// TIA Portal project "DPS" (V18)

(* hardware
DEVICE "S7-1200-Station_1"  S7-1200 Station
   slot 0: "Baugruppenträger_0"  S7-1200 Rack  Rack  V1.0
   slot 1: "DPS"  CPU 1215C DC/DC/DC  6ES7 215-1AG40-0XB0  V4.5
*)

// ===== PLC "DPS"  CPU 1215C DC/DC/DC =====

VAR_GLOBAL   // PLC tag table "Lichter"
   "grünLED" AT %Q0.4 : Bool;
   "gelbLED" AT %Q0.5 : Bool;
   "rotLED" AT %Q0.6 : Bool;
   "rotLED_online" AT %Q0.7 : Bool;
END_VAR

VAR_GLOBAL   // PLC tag table "Farbsensor"
   "FarbWert" AT %IW64 : Int;
END_VAR

VAR_GLOBAL   // PLC tag table "WareneingangAusgang"
   "ausgangLS" AT %I0.2 : Bool;
   "eingangLS" AT %I0.3 : Bool;
END_VAR

VAR_GLOBAL   // PLC tag table "KameraHR"
   "refKameraHochRunter" AT %I0.0 : Bool;   // Referenzschalter für den Encoder
   "encoderHR_A" AT %I0.4 : Bool;   // Encoder A
   "encoderHR_B" AT %I0.5 : Bool;   // Encoder B
   "kameraHoch" AT %Q0.0 : Bool;   // Motor drehen um Kamera nach oben zu bewegen
   "kameraRunter" AT %Q0.1 : Bool;   // Motor drehen um Kamera nach unten zu bewegen
   "PWM_kameraHR" AT %QW1000 : Int;   // Prozentualer Wert für die geschwindigkeit des Motors
   "EncoderWertHR" AT %ID1000 : DInt;   // Der Zählwert welche die Position bestimmt
END_VAR

VAR_GLOBAL   // PLC tag table "KameraLR"
   "refKameraLinksRechts" AT %I0.1 : Bool;   // Referenzschalter für den Encoder
   "encoderLR_A" AT %I0.6 : Bool;   // Encoder A
   "encoderLR_B" AT %I0.7 : Bool;   // Encoder B
   "kameraLinks" AT %Q0.2 : Bool;   // Motor drehen um Kamera nach links zu bewegen
   "kameraRechts" AT %Q0.3 : Bool;   // Motor drehen um Kamera nach rechts zu bewegen
   "PWM_kameraLR" AT %QW1002 : Int;   // Prozentualer Wert für die geschwindigkeit des Motors
   "EncoderWertLR" AT %ID1004 : DInt;   // Der Zählwert welche die Position bestimmt
END_VAR

DATA_BLOCK "DB_Global"   // DB1
{ S7_Optimized_Access := 'TRUE' }
VERSION : 0.1
   VAR
      farbwert : Int;
      farbbereich_rot : Bool;
      farbbereich_weiss : Bool;
      farbbereich_blau : Bool;
      input : Bool;
      output : Bool;
      referenziert_X : Bool;
      referenziert_Y : Bool;
      referenzieren : Bool;
      reset : Bool;
      Farbe : Struct
         berechne : Bool;
         rotOben : Int;
         rotUnten : Int;
         weissOben : Int;
         weissUnten : Int;
         blauOben : Int;
         blauUnten : Int;
      END_STRUCT;
   END_VAR
BEGIN
END_DATA_BLOCK

DATA_BLOCK "DB_Referenzen"   // DB2
{ S7_Optimized_Access := 'TRUE' }
VERSION : 0.1
   VAR RETAIN
      Calib : Struct
         Limits : Struct
            grenze_x_oben : DInt := 1700;
            grenze_x_unten : DInt := 0;
            grenze_y_oben : DInt := 700;
            grenze_y_unten : DInt := 0;
         END_STRUCT;
         Positionen : Struct
            Home : Struct
               position_home_X : DInt := 900;
               position_home_Y : DInt := 350;
            END_STRUCT;
            HBW : Struct
               position_hbw_X : DInt := 1500;
               position_hbw_Y : DInt := 250;
            END_STRUCT;
            Parken : Struct
               position_parken_X : DInt := 1000;
               position_parken_Y : DInt := 5;
            END_STRUCT;
         END_STRUCT;
         Farbe : Struct
            farbe_rot_richtwert : Int := 17500;
            farbe_blau_richtwert : Int := 20500;
            farbe_weiss_richtwert : Int := 6300;
            farbe_wertbereich : Int := 1500;
         END_STRUCT;
         zeit_prozessWarteZeitKurz : Time := T#500MS;
      END_STRUCT;
      Defaults : Struct
         Limits : Struct
            grenze_x_oben : DInt := 1700;
            grenze_x_unten : DInt := 0;
            grenze_y_oben : DInt := 700;
            grenze_y_unten : DInt := 0;
         END_STRUCT;
         Positionen : Struct
            Home : Struct
               position_home_X : DInt := 900;
               position_home_Y : DInt := 350;
            END_STRUCT;
            HBW : Struct
               position_hbw_X : DInt := 1500;
               position_hbw_Y : DInt := 250;
            END_STRUCT;
         END_STRUCT;
         Farbe : Struct
            farbe_rot_richtwert : Int := 17500;
            farbe_blau_richtwert : Int := 20500;
            farbe_weiss_richtwert : Int := 6300;
            farbe_wertbereich : Int := 1500;
         END_STRUCT;
         zeit_prozessWarteZeitKurz : Time := T#500MS;
      END_STRUCT;
      bereich_langsam : DInt := 5;
      genauigkeit : DInt := 1;
      PWM_langsam : DInt := 50;
      PWM_schnell : DInt := 100;
      model : String := 'DPS';
   END_VAR
   VAR
      "version" : String := '1.5.0';
   END_VAR
BEGIN
END_DATA_BLOCK

DATA_BLOCK "FB_OrderOrganisation_DB"   // DB3
{ S7_Optimized_Access := 'TRUE' }
VERSION : 0.1
// stored: InstanceOfName FB_OrderOrganisation
"FB_OrderOrganisation"
BEGIN
END_DATA_BLOCK

DATA_BLOCK "FB_Kalibrierung_DB"   // DB4
{ S7_Optimized_Access := 'TRUE' }
VERSION : 0.1
// stored: InstanceOfName FB_Kalibrierung
"FB_Kalibrierung"
BEGIN
END_DATA_BLOCK

// folder: Encoder

DATA_BLOCK "FB_Positionierung_DB"   // DB7
{ S7_Optimized_Access := 'TRUE' }
VERSION : 0.1
// stored: InstanceOfName FB_Positionierung
"FB_Positionierung"
BEGIN
END_DATA_BLOCK

// folder: (top level)

FUNCTION_BLOCK "FB_OrderOrganisation"   // FB1, FBD
{ S7_Optimized_Access := 'TRUE' }
VERSION : 0.1
   VAR
      Lampe : Struct
         lampe_onlineROT : Bool;
         lampe_ROT : Bool;
         lampe_GELB : Bool;
         lampe_GRÜN : Bool;
      END_STRUCT;
      Befehle : Struct
         befehl_BEWEGEN : Bool;
         bewegen_aktiv : Bool;
         bewegen_finished : Bool;
         bewegen_position_X : DInt;
         bewegen_position_Y : DInt;
         befehl_HOME : Bool;
         home_aktiv : Bool;
         home_finished : Bool;
         befehl_HBW : Bool;
         hbw_aktiv : Bool;
         hbw_finished : Bool;
         befehl_KALIBRIERE : Bool;
         kalibriere_aktiv : Bool;
         kalibriere_finished : Bool;
      END_STRUCT;
      "step" : DInt;
      busy : Bool;
      warten : TON_TIME;
      wartenZeit : Time;
      wartenStart : Bool;
   END_VAR
BEGIN

REGION Network 1: Timer
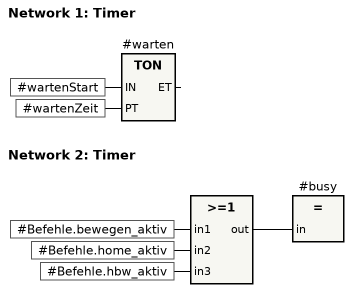
   #warten(IN := #wartenStart, PT := #wartenZeit);   // TON
END_REGION

REGION Network 2: Timer
   #busy := #Befehle.bewegen_aktiv OR #Befehle.home_aktiv OR #Befehle.hbw_aktiv;
END_REGION

REGION Network 3 (SCL): Ablauf
   // Befehle:
   // Fahre auf position
   // Kamera auf Home
   // Kamera auf HBW (Variable Position)


   CASE #step OF
       0: // Init
           IF "DB_Global".referenziert_X AND "DB_Global".referenziert_Y THEN
               #step := 2;
           END_IF
           ;
       1: // Befehl 
           // mehrfachaufruf verhindern
           #Befehle.befehl_KALIBRIERE := FALSE;
           // Farbegrenzen aktualisieren
           "DB_Global".Farbe.berechne := TRUE;
           // finished zurücksetzen
           #Befehle.kalibriere_finished := FALSE;
           #Befehle.bewegen_finished := FALSE;
           #Befehle.home_finished := FALSE;
           #Befehle.hbw_finished := FALSE;
           #step := 4
           ;
       2: // Home Position anfahren

           // Werte aktualisieren
           #Befehle.bewegen_position_X := "DB_Referenzen".Calib.Positionen.Home.position_home_X;
           #Befehle.bewegen_position_Y := "DB_Referenzen".Calib.Positionen.Home.position_home_Y;

           "FB_Positionierung_DB".Achsen.X.sollPosition := "DB_Referenzen".Calib.Positionen.Home.position_home_X;
           "FB_Positionierung_DB".Achsen.Y.sollPosition := "DB_Referenzen".Calib.Positionen.Home.position_home_Y;
           // Positionierung Starten
           "FB_Positionierung_DB".finished := FALSE;
           "FB_Positionierung_DB".startPositionierung := TRUE;
           #step := 3;
       3: // warte auf Ende Positionierung
           IF "FB_Positionierung_DB".finished THEN
               #step := 1;
           END_IF
           ;
       4:  // warten auf FLAG busy
           IF NOT #busy THEN
               #step := 5;
           END_IF
           ;
       5: // Bereit für KameraBefehle
           IF #Befehle.befehl_BEWEGEN THEN
               #Befehle.befehl_BEWEGEN := FALSE;
               #Befehle.bewegen_aktiv := TRUE;
               #step := 10;
           ELSIF #Befehle.befehl_HBW THEN
               #Befehle.befehl_HBW := FALSE;
               #Befehle.hbw_aktiv := TRUE;
               #step := 50;
           ELSIF #Befehle.befehl_HOME THEN
               #Befehle.befehl_HOME := FALSE;
               #Befehle.home_aktiv := TRUE;
               #step := 100;
           ELSIF #Befehle.befehl_KALIBRIERE THEN
               #Befehle.befehl_KALIBRIERE := FALSE;
               #Befehle.kalibriere_aktiv := TRUE;
               #step := 150;
           END_IF
           ;
           "DB_Global".Farbe.berechne := FALSE;
       10: // Positionen übergeben ------------------------- Fahre Position an
           "FB_Positionierung_DB".Achsen.X.sollPosition := #Befehle.bewegen_position_X;
           "FB_Positionierung_DB".Achsen.Y.sollPosition := #Befehle.bewegen_position_Y;
           // Positionierung Starten
           "FB_Positionierung_DB".finished := FALSE;
           "FB_Positionierung_DB".startPositionierung := TRUE;
           #step := 11
           ;
       11: // warte auf Ende Positionierung
           IF "FB_Positionierung_DB".finished THEN
               #step := 12;
           END_IF
           ;
       12: // Flag finished setzen
           #Befehle.bewegen_finished := TRUE;
           #step := 13;
       13: // kurz warten
           #wartenZeit := "DB_Referenzen".Calib.zeit_prozessWarteZeitKurz;
           #wartenStart := TRUE;
           IF #warten.Q THEN
               #Befehle.bewegen_aktiv := FALSE;
               #wartenStart := FALSE;
               #step := 1;
           END_IF
           ;

       50: // Positionen übergeben ------------------------- Fahre HBW an

           // Werte aktualisieren
           #Befehle.bewegen_position_X := "DB_Referenzen".Calib.Positionen.HBW.position_hbw_X;
           #Befehle.bewegen_position_Y := "DB_Referenzen".Calib.Positionen.HBW.position_hbw_Y;

           "FB_Positionierung_DB".Achsen.X.sollPosition := "DB_Referenzen".Calib.Positionen.HBW.position_hbw_X;
           "FB_Positionierung_DB".Achsen.Y.sollPosition := "DB_Referenzen".Calib.Positionen.HBW.position_hbw_Y;
           // Positionierung Starten
           "FB_Positionierung_DB".finished := FALSE;
           "FB_Positionierung_DB".startPositionierung := TRUE;
           #step := 51
           ;
       51: // warte auf Ende Positionierung
           IF "FB_Positionierung_DB".finished THEN
               #step := 52;
           END_IF
           ;
       52: // Flag finished setzen
           #Befehle.hbw_finished := TRUE;
           #step := 53;
       53: // kurz warten
           #wartenZeit := "DB_Referenzen".Calib.zeit_prozessWarteZeitKurz;
           #wartenStart := TRUE;
           IF #warten.Q THEN
               #Befehle.hbw_aktiv := FALSE;
               #wartenStart := FALSE;
               #step := 1;
           END_IF
           ;
       100: // Positionen übergeben ------------------------- Fahre Home an

           // Werte aktualisieren
           #Befehle.bewegen_position_X := "DB_Referenzen".Calib.Positionen.Home.position_home_X;
           #Befehle.bewegen_position_Y := "DB_Referenzen".Calib.Positionen.Home.position_home_Y;

           "FB_Positionierung_DB".Achsen.X.sollPosition := "DB_Referenzen".Calib.Positionen.Home.position_home_X;
           "FB_Positionierung_DB".Achsen.Y.sollPosition := "DB_Referenzen".Calib.Positionen.Home.position_home_Y;
           // Positionierung Starten
           "FB_Positionierung_DB".finished := FALSE;
           "FB_Positionierung_DB".startPositionierung := TRUE;
           #step := 101
           ;
       101: // warte auf beendung
           IF "FB_Positionierung_DB".finished THEN
               #step := 102;
           END_IF
           ;
       102: // Flag finished setzen
           #Befehle.home_finished := TRUE;
           #step := 103;
       103: // kurz warte für NodeRed
           #wartenZeit := "DB_Referenzen".Calib.zeit_prozessWarteZeitKurz;
           #wartenStart := TRUE;
           IF #warten.Q THEN
               #Befehle.home_aktiv := FALSE;
               #wartenStart := FALSE;
               #step := 1;
           END_IF
           ;
       150: // Auf ende Kalibrierung warten
           IF NOT #Befehle.kalibriere_aktiv AND #Befehle.kalibriere_finished THEN
               #step := 151;
           END_IF
           ;
       151: // warten
           #wartenZeit := "DB_Referenzen".Calib.zeit_prozessWarteZeitKurz;
           #wartenStart := TRUE;
           IF #warten.Q THEN
               #step := 1;
           END_IF
           ;


           ELSE  // Statement section ELSE
               ;
   END_CASE;
END_REGION
END_FUNCTION_BLOCK

FUNCTION_BLOCK "FB_Kalibrierung"   // FB2, FBD
{ S7_Optimized_Access := 'TRUE' }
VERSION : 0.1
   VAR
      befehl_DEFAULT : Bool;
      default_finished : Bool;
      befehl_ANFAHREN : Bool;
      anfahren_position_X : DInt;
      anfahren_position_Y : DInt;
      anfahren_finished : Bool;
      befehl_BEENDEN : Bool;
      beenden_finished : Bool;
      "step" : DInt;
      warten : TON_TIME;
      wartenStart : Bool;
      wartenZeit : Time;
      befehl_PARKEN : Bool;
      parken_aktiv : Bool;
   END_VAR
BEGIN

REGION Network 1
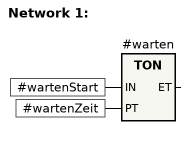
   #warten(IN := #wartenStart, PT := #wartenZeit);   // TON
END_REGION

REGION Network 2 (SCL)
   CASE #step OF
       0: // init
           #step := 1
           ;
       1: // Befehle und flags FALSE setzen
           #befehl_PARKEN := FALSE;
           #default_finished := FALSE;
           #anfahren_finished := FALSE;
           #beenden_finished := FALSE;
           #befehl_DEFAULT := FALSE;
           #befehl_ANFAHREN := FALSE;
           #befehl_BEENDEN := FALSE;
           #step := 2
           ;
       2: // Kalib check    
           IF "FB_OrderOrganisation_DB".Befehle.kalibriere_aktiv THEN
               #step := 3;
           END_IF
           ;
       3: // Auf Befehle warten

           IF #befehl_BEENDEN THEN
               #step := 100;
           ELSIF #befehl_ANFAHREN THEN
               #step := 10;
           ELSIF #befehl_DEFAULT THEN
               #step := 50;
           ELSIF #befehl_PARKEN THEN
               #step := 20;
           END_IF
           ;
       10: // übergebe Positionen
           "FB_Positionierung_DB".Achsen.X.sollPosition := #anfahren_position_X;
           "FB_Positionierung_DB".Achsen.Y.sollPosition := #anfahren_position_Y;

           // positionerung starten
           "FB_Positionierung_DB".finished := FALSE;
           "FB_Positionierung_DB".startPositionierung := TRUE;

           #step := 11
           ;
       11: // warten auf Ende Positionierung
           IF "FB_Positionierung_DB".finished THEN
               #step := 12;
           END_IF
           ;
       12: // setze auf finished
           IF #parken_aktiv THEN
               #parken_aktiv := FALSE;
           END_IF;
           #anfahren_finished := TRUE;
           #wartenZeit := "DB_Referenzen".Calib.zeit_prozessWarteZeitKurz;
           #wartenStart := TRUE;
           IF #warten.Q THEN
               #wartenStart := FALSE;
               #step := 1;
           END_IF
           ;
       20: // Parken
           #parken_aktiv := TRUE;
           // positionen übergeben
           #anfahren_position_X := "DB_Referenzen".Calib.Positionen.Parken.position_parken_X;
           #anfahren_position_Y := "DB_Referenzen".Calib.Positionen.Parken.position_parken_Y;
           #step := 21
           ;
       21: // weiter zu anfahren
           #step := 10
           ;
       50: // Werte auf Default zurücksetzen
           "DB_Referenzen".Calib.Limits.grenze_x_oben := "DB_Referenzen".Defaults.Limits.grenze_x_oben;
           "DB_Referenzen".Calib.Limits.grenze_x_unten := "DB_Referenzen".Defaults.Limits.grenze_x_unten;
           "DB_Referenzen".Calib.Limits.grenze_y_oben := "DB_Referenzen".Defaults.Limits.grenze_y_oben;
           "DB_Referenzen".Calib.Limits.grenze_y_unten := "DB_Referenzen".Defaults.Limits.grenze_y_unten;

           "DB_Referenzen".Calib.Positionen.Home.position_home_X := "DB_Referenzen".Defaults.Positionen.Home.position_home_X;
           "DB_Referenzen".Calib.Positionen.Home.position_home_Y := "DB_Referenzen".Defaults.Positionen.Home.position_home_Y;

           "DB_Referenzen".Calib.Positionen.HBW.position_hbw_X := "DB_Referenzen".Defaults.Positionen.HBW.position_hbw_X;
           "DB_Referenzen".Calib.Positionen.HBW.position_hbw_Y := "DB_Referenzen".Defaults.Positionen.HBW.position_hbw_Y;

           "DB_Referenzen".Calib.Farbe.farbe_rot_richtwert := "DB_Referenzen".Defaults.Farbe.farbe_rot_richtwert;
           "DB_Referenzen".Calib.Farbe.farbe_blau_richtwert := "DB_Referenzen".Defaults.Farbe.farbe_blau_richtwert;
           "DB_Referenzen".Calib.Farbe.farbe_weiss_richtwert := "DB_Referenzen".Defaults.Farbe.farbe_weiss_richtwert;

           "DB_Referenzen".Calib.zeit_prozessWarteZeitKurz := "DB_Referenzen".Defaults.zeit_prozessWarteZeitKurz;

           #step := 51
           ;
       51: // kurz warten
           #wartenZeit := "DB_Referenzen".Calib.zeit_prozessWarteZeitKurz;
           #wartenStart := TRUE;
           IF #warten.Q THEN
               #wartenStart := FALSE;
               #step := 1;
           END_IF
           ;
       100: // Beenden der Kalibrierung
           // Farbgrenzen berechnen
           "DB_Global".Farbe.berechne := TRUE;

           // status setzen
           "FB_OrderOrganisation_DB".Befehle.kalibriere_finished := TRUE;
           "FB_OrderOrganisation_DB".Befehle.kalibriere_aktiv := FALSE;
           #step := 101
           ;
       101: // prozess Ende
           #wartenZeit := "DB_Referenzen".Calib.zeit_prozessWarteZeitKurz;
           #wartenStart := TRUE;
           IF #warten.Q THEN
               #wartenStart := FALSE;
               #step := 1;
           END_IF
           ;
       ELSE 
           ;
   END_CASE;
END_REGION
END_FUNCTION_BLOCK

FUNCTION "FC_Referenzieren" : Void   // FC1, FBD
{ S7_Optimized_Access := 'TRUE' }
VERSION : 0.1
BEGIN

REGION Network 1: PWM für HBW schreiben
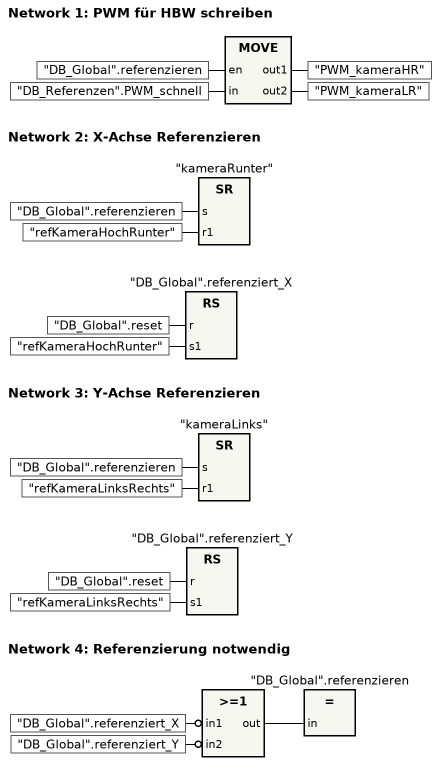
   IF "DB_Global".referenzieren THEN
       "PWM_kameraHR" := "DB_Referenzen".PWM_schnell;
       "PWM_kameraLR" := "DB_Referenzen".PWM_schnell;
   END_IF;
END_REGION

REGION Network 2: X-Achse Referenzieren
   IF "DB_Global".referenzieren THEN
       "kameraRunter" := TRUE;   // SR flip-flop
   END_IF;
   IF "refKameraHochRunter" THEN "kameraRunter" := FALSE; END_IF;
   IF "DB_Global".reset THEN
       "DB_Global".referenziert_X := FALSE;   // RS flip-flop
   END_IF;
   IF "refKameraHochRunter" THEN "DB_Global".referenziert_X := TRUE; END_IF;
END_REGION

REGION Network 3: Y-Achse Referenzieren
   IF "DB_Global".referenzieren THEN
       "kameraLinks" := TRUE;   // SR flip-flop
   END_IF;
   IF "refKameraLinksRechts" THEN "kameraLinks" := FALSE; END_IF;
   IF "DB_Global".reset THEN
       "DB_Global".referenziert_Y := FALSE;   // RS flip-flop
   END_IF;
   IF "refKameraLinksRechts" THEN "DB_Global".referenziert_Y := TRUE; END_IF;
END_REGION

REGION Network 4: Referenzierung notwendig
   "DB_Global".referenzieren := NOT "DB_Global".referenziert_X OR NOT "DB_Global".referenziert_Y;
END_REGION
END_FUNCTION

FUNCTION "FC_Verwaltung" : Void   // FC2, FBD
{ S7_Optimized_Access := 'TRUE' }
VERSION : 0.1
   VAR_TEMP
      blau_rot_grenze : Int;
      rot_weiss_grenze : Int;
   END_VAR
BEGIN

REGION Network 1: PWM Kamera Hoch Runter
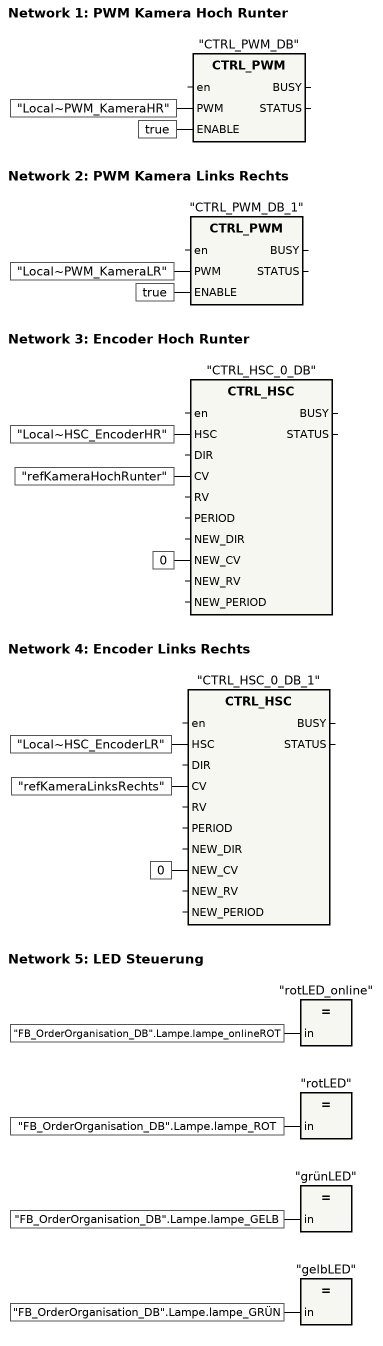
   "CTRL_PWM_DB"(PWM := "Local~PWM_KameraHR", ENABLE := true);   // CTRL_PWM
END_REGION

REGION Network 2: PWM Kamera Links Rechts
   "CTRL_PWM_DB_1"(PWM := "Local~PWM_KameraLR", ENABLE := true);   // CTRL_PWM
END_REGION

REGION Network 3: Encoder Hoch Runter
   "CTRL_HSC_0_DB"(HSC := "Local~HSC_EncoderHR", CV := "refKameraHochRunter", NEW_CV := 0);   // CTRL_HSC
END_REGION

REGION Network 4: Encoder Links Rechts
   "CTRL_HSC_0_DB_1"(HSC := "Local~HSC_EncoderLR", CV := "refKameraLinksRechts", NEW_CV := 0);   // CTRL_HSC
END_REGION

REGION Network 5: LED Steuerung
   "rotLED_online" := "FB_OrderOrganisation_DB".Lampe.lampe_onlineROT;
   "rotLED" := "FB_OrderOrganisation_DB".Lampe.lampe_ROT;
   "grünLED" := "FB_OrderOrganisation_DB".Lampe.lampe_GELB;
   "gelbLED" := "FB_OrderOrganisation_DB".Lampe.lampe_GRÜN;
END_REGION

REGION Network 6: Input / Output Lichtschranke
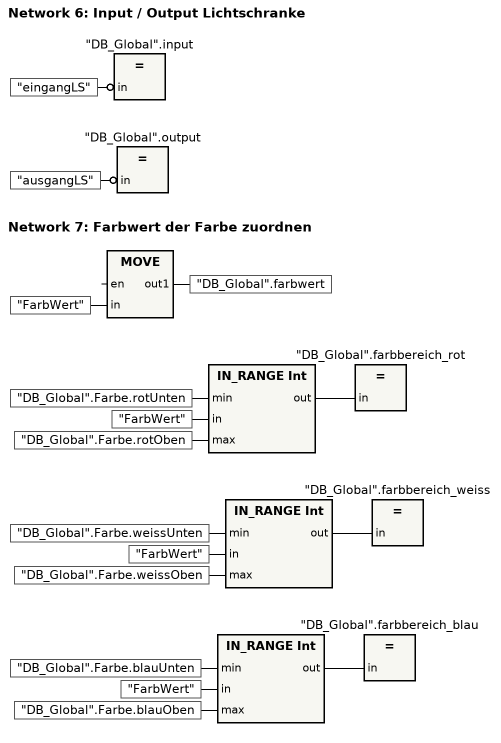
   "DB_Global".input := NOT "eingangLS";
   "DB_Global".output := NOT "ausgangLS";
END_REGION

REGION Network 7: Farbwert der Farbe zuordnen
   "DB_Global".farbwert := "FarbWert";
   "DB_Global".farbbereich_rot := ("DB_Global".Farbe.rotUnten <= "FarbWert") AND ("FarbWert" <= "DB_Global".Farbe.rotOben);
   "DB_Global".farbbereich_weiss := ("DB_Global".Farbe.weissUnten <= "FarbWert") AND ("FarbWert" <= "DB_Global".Farbe.weissOben);
   "DB_Global".farbbereich_blau := ("DB_Global".Farbe.blauUnten <= "FarbWert") AND ("FarbWert" <= "DB_Global".Farbe.blauOben);
END_REGION

REGION Network 8 (SCL): Berechnung der Farbgrenzen
   // Berechnung der Farbwerte

   // Recalculate color boundaries from config
   IF "DB_Global".Farbe.berechne THEN

       // Absolute upper and lower boundaries
       "DB_Global".Farbe.blauOben := 32767;
       "DB_Global".Farbe.weissUnten := 0;

       // Boundary between blue and red
       #blau_rot_grenze := ("DB_Referenzen".Calib.Farbe.farbe_blau_richtwert - "DB_Referenzen".Calib.Farbe.farbe_rot_richtwert) / 2;
       "DB_Global".Farbe.rotOben := "DB_Referenzen".Calib.Farbe.farbe_rot_richtwert + #blau_rot_grenze;
       "DB_Global".Farbe.blauUnten :=  "DB_Referenzen".Calib.Farbe.farbe_blau_richtwert - #blau_rot_grenze + 1;

       // Boundary between white and red
       #rot_weiss_grenze := ("DB_Referenzen".Calib.Farbe.farbe_rot_richtwert - "DB_Referenzen".Calib.Farbe.farbe_weiss_richtwert) / 2;
       "DB_Global".Farbe.rotUnten := "DB_Referenzen".Calib.Farbe.farbe_rot_richtwert - #rot_weiss_grenze + 1;
       "DB_Global".Farbe.weissOben := "DB_Referenzen".Calib.Farbe.farbe_weiss_richtwert + #rot_weiss_grenze;
   END_IF;
END_REGION
END_FUNCTION

ORGANIZATION_BLOCK "Main"   // OB1, FBD, ProgramCycle
TITLE = "Main Program Sweep (Cycle)"
{ S7_Optimized_Access := 'TRUE' }
VERSION : 0.1
   VAR_INPUT
      Initial_Call : Bool;   // Initial call of this OB
      Remanence : Bool;   // =True, if remanent data are available
   END_VAR
BEGIN

REGION Network 1: Verwaltung
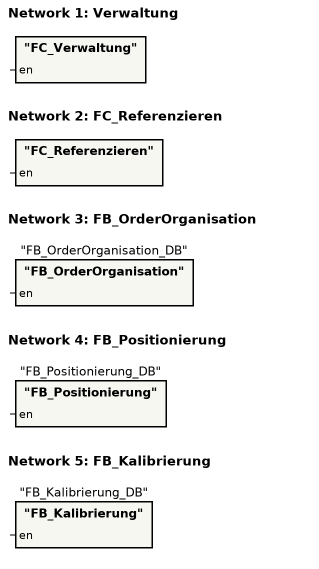
   "FC_Verwaltung"();
END_REGION

REGION Network 2: FC_Referenzieren
   "FC_Referenzieren"();
END_REGION

REGION Network 3: FB_OrderOrganisation
   "FB_OrderOrganisation_DB"();   // "FB_OrderOrganisation"
END_REGION

REGION Network 4: FB_Positionierung
   "FB_Positionierung_DB"();   // "FB_Positionierung"
END_REGION

REGION Network 5: FB_Kalibrierung
   "FB_Kalibrierung_DB"();   // "FB_Kalibrierung"
END_REGION
END_ORGANIZATION_BLOCK

// folder: Encoder

FUNCTION_BLOCK "FB_Positionierung"   // FB3, FBD
TITLE = Positionierung
{ S7_Optimized_Access := 'TRUE' }
// Der Baustein muss im Main dauerhaft an sein um richtig zu funktionieren
// 
// Bevor die Variable "startPositionierung" TRUE und "finished" FALSE gesetzt werden.
// Die "Sollpositionen" sind genauso müssen auch übertragen worden sein bevor die startPositionierung TRUE gesetzt wird.
// 
// "finished" wird vom Baustein wieder TRUE gesetzt wenn, alle 3 Achsen die Position erreicht haben.
   VAR
      startPositionierung : Bool;
      working : Bool;
      finished : Bool;
      Achsen : Struct
         X : Struct
            sollPosition : DInt;
            start : Bool;
            positionErreicht : Bool;
         END_STRUCT;
         Y : Struct
            sollPosition : DInt;
            start : Bool;
            positionErreicht : Bool;
         END_STRUCT;
      END_STRUCT;
      "step" : DInt;
      zuGroßX : Bool;
      zuKleinX : Bool;
      zuGroßY : Bool;
      zuKleinY : Bool;
   END_VAR
BEGIN

REGION Network 1 (SCL): Schrittkette
   CASE #step OF
       0:  // Start Positionierung
           IF #startPositionierung AND NOT #working THEN
               #startPositionierung := FALSE;
               #working := TRUE;
               #step := 1;
           END_IF
           ;
       1: // check ob variablen außerhalb der Limits ist
           // X-Achse
           IF #zuGroßX THEN
               #Achsen.X.sollPosition := "DB_Referenzen".Calib.Limits.grenze_x_oben
               ;
           ELSIF #zuKleinX THEN
               #Achsen.X.sollPosition := "DB_Referenzen".Calib.Limits.grenze_x_unten
               ;
           END_IF
           ;
           // Y-Achse
           IF #zuGroßY THEN
               #Achsen.Y.sollPosition := "DB_Referenzen".Calib.Limits.grenze_y_oben
               ;
           ELSIF #zuKleinY THEN
               #Achsen.Y.sollPosition := "DB_Referenzen".Calib.Limits.grenze_y_unten
               ;
           END_IF
           ;
           #step := 2;
       2:  // Starte Achsen
           #Achsen.X.positionErreicht := FALSE;
           #Achsen.Y.positionErreicht := FALSE;


           #Achsen.X.start := TRUE;
           #Achsen.Y.start := TRUE;


           #step := 10;

       10:  // Stoppe Achsen
           IF #Achsen.X.positionErreicht THEN
               #Achsen.X.start := FALSE;
           END_IF;

           IF #Achsen.Y.positionErreicht THEN
               #Achsen.Y.start := FALSE;
           END_IF;

           IF #Achsen.X.positionErreicht AND #Achsen.Y.positionErreicht THEN
               #step := 20;
           END_IF
           ;
       20: // 
           #working := FALSE;
           #finished := TRUE;
           #step := 0
           ;
       ELSE  // Statement section ELSE
           ;
   END_CASE;
END_REGION

REGION Network 2: Positionierung X Links Rechts
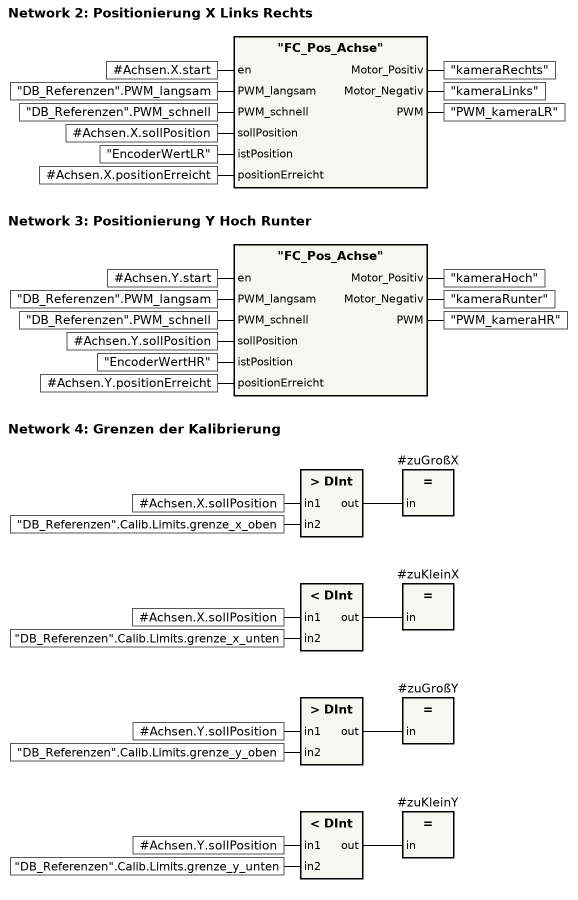
   IF #Achsen.X.start THEN
       "FC_Pos_Achse"(PWM_langsam := "DB_Referenzen".PWM_langsam,
                      PWM_schnell := "DB_Referenzen".PWM_schnell,
                      sollPosition := #Achsen.X.sollPosition,
                      istPosition := "EncoderWertLR",
                      positionErreicht := #Achsen.X.positionErreicht,
                      Motor_Positiv => "kameraRechts",
                      Motor_Negativ => "kameraLinks",
                      PWM => "PWM_kameraLR");
   END_IF;
END_REGION

REGION Network 3: Positionierung Y Hoch Runter
   IF #Achsen.Y.start THEN
       "FC_Pos_Achse"(PWM_langsam := "DB_Referenzen".PWM_langsam,
                      PWM_schnell := "DB_Referenzen".PWM_schnell,
                      sollPosition := #Achsen.Y.sollPosition,
                      istPosition := "EncoderWertHR",
                      positionErreicht := #Achsen.Y.positionErreicht,
                      Motor_Positiv => "kameraHoch",
                      Motor_Negativ => "kameraRunter",
                      PWM => "PWM_kameraHR");
   END_IF;
END_REGION

REGION Network 4: Grenzen der Kalibrierung
   #zuGroßX := #Achsen.X.sollPosition > "DB_Referenzen".Calib.Limits.grenze_x_oben;
   #zuKleinX := #Achsen.X.sollPosition < "DB_Referenzen".Calib.Limits.grenze_x_unten;
   #zuGroßY := #Achsen.Y.sollPosition > "DB_Referenzen".Calib.Limits.grenze_y_oben;
   #zuKleinY := #Achsen.Y.sollPosition < "DB_Referenzen".Calib.Limits.grenze_y_unten;
END_REGION
END_FUNCTION_BLOCK

FUNCTION "FC_Pos_Achse" : Void   // FC9, FBD
{ S7_Optimized_Access := 'TRUE' }
   VAR_INPUT
      PWM_langsam : DInt;
      PWM_schnell : DInt;
      sollPosition : DInt;
      istPosition : DInt;
   END_VAR
   VAR_OUTPUT
      Motor_Positiv : Bool;
      Motor_Negativ : Bool;
      PWM : DInt;
   END_VAR
   VAR_IN_OUT
      positionErreicht : Bool;
   END_VAR
   VAR_TEMP
      langsamOben : DInt;
      langsamUnten : DInt;
      grenzeOben : DInt;
      grenzeUnten : DInt;
   END_VAR
   VAR_TEMP   // added for the SCL form of the ladder/FBD networks
      _w1 : Bool;
   END_VAR
BEGIN

REGION Network 1: Berechne Grenzen X
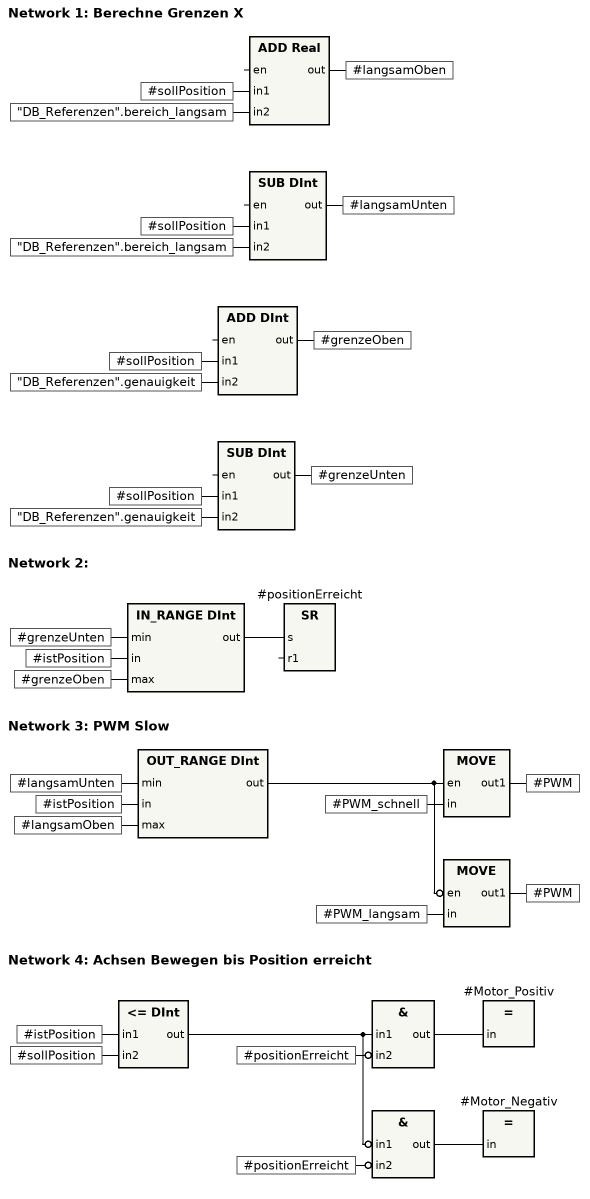
   #langsamOben := #sollPosition + "DB_Referenzen".bereich_langsam;
   #langsamUnten := #sollPosition - "DB_Referenzen".bereich_langsam;
   #grenzeOben := #sollPosition + "DB_Referenzen".genauigkeit;
   #grenzeUnten := #sollPosition - "DB_Referenzen".genauigkeit;
END_REGION

REGION Network 2
   IF (#grenzeUnten <= #istPosition) AND (#istPosition <= #grenzeOben) THEN
       #positionErreicht := TRUE;   // SR flip-flop
   END_IF;
END_REGION

REGION Network 3: PWM Slow
   #_w1 := (#istPosition < #langsamUnten) OR (#istPosition > #langsamOben);
   IF #_w1 THEN #PWM := #PWM_schnell; END_IF;
   IF NOT #_w1 THEN #PWM := #PWM_langsam; END_IF;
END_REGION

REGION Network 4: Achsen Bewegen bis Position erreicht
   #_w1 := #istPosition <= #sollPosition;
   #Motor_Positiv := #_w1 AND NOT #positionErreicht;
   #Motor_Negativ := NOT #_w1 AND NOT #positionErreicht;
END_REGION
END_FUNCTION